TYPE CmpWorkStopMainLnSw :
STRUCT
	Framework: Framework;
	Config: CmpWorkStopMainLnSwConfig;
	Sim: CmpWorkStopMainLnSwSim;
	WorkReq: BOOL;
	WorkCmp: BOOL;
	PuckLnSw: PuckLnSw;
	DevicePresent: BOOL;
END_STRUCT
END_TYPE

(* stored: Version 1.1.0.1, ProductVersion 3.1.4024.6
   DUT CmpWorkStopMainLnSw: Id {e36249a3-f0c3-4549-8662-31e24a1aedcc} *)
